{attribute addProperty BoxType "EL1262-0000-0002"}
{attribute addProperty Id "Ch2_InputAT %I*BOOL81"}
{attribute addProperty CRC "3820424950"}
{attribute addProperty SizeInBites "8"}
{attribute addProperty SizeInBytes "1"}
TYPE Ch2_Input_E3B70EF6 :
STRUCT
	{attribute addProperty Name "Ch2_Input"}
	Ch2_Input AT %I* : BOOL;
END_STRUCT
END_TYPE

(* stored: Version 1.2.0.0, ProductVersion 3.1.4024.9
   DUT Ch2_Input_E3B70EF6: Id {812f6b37-e0ba-49ac-9835-4568135aa2a9} *)
